PROGRAM MAIN
VAR
	t_startTimeRt AT %I* :ULINT; 
	rtStartTime : TIMESTRUCT;
	b_convert : BOOL;
END_VAR

IF b_convert THEN
	rtStartTime := DT_TO_SYSTEMTIME(FILETIME64_TO_DT(t_startTimeRt));
END_IF

END_PROGRAM

(* stored: Version 1.1.0.1, ProductVersion 3.1.4024.12
   POU MAIN: Id {3c5d083f-b959-44bc-acb3-e333f358aaea}, SpecialFunc None *)
